# EPICS SNL sequencer program: kstar/siteApp/DLS/DLSApp/src/sncDlsTSE.stt
program sncDlsTSE
option +r;
option +c;
%% #include <string.h>
%% #include <epicsPrint.h>

int status;
int close;
int open;

%% /* PV name Changed DLS_THOMSONEDGE_N_OP_SHUT, DLS_THOMSONEDGE_N_CL_SHUT  */

assign status to "DLS_THOMSONEDGE_N_SHUT_STATUS";
monitor status;

assign close to "DLS_THOMSONEDGE_N_SHUT_CLOSE_READ";
monitor close;
assign open to "DLS_THOMSONEDGE_N_SHUT_OPEN_READ";
monitor open;

ss dlsTSEStatus{
	state init{
		when (TRUE){
			if(close==1 && open ==0) {
				status=0;
				pvPut(status);
			} else if(close==0 && open==1) {
				status=1;
				pvPut(status);
			} else if(close==0 && open==0) {
				status=2;
				pvPut(status);
			} else if(close==1 && open ==1) {
				status=3;
                                pvPut(status);
			}
		}state dls_check
	}
	state dls_check {
        	when (delay(1.0)){
			if(close==1 && open ==0) {
				status=0;
				pvPut(status);
			} else if(close==0 && open==1) {
				status=1;
				pvPut(status);
			} else if(close==0 && open==0) {
				status=2;
				pvPut(status);
			} else if(close==1 && open ==1) {
				status=3;
                                pvPut(status);
			}
		} state dls_check
	}
}
